(* CODESYS project Automatic stacking program.project

Project tree, tasks and I/O mapping:
  Device : CODESYS Control Win V3, 3S - Smart Software Solutions GmbH, order no. 305021, version 3.5.7.0
    application Application
      libraries: Standard, * (System)
      task MainTask (cyclic, interval t#20ms, priority 1) calls PLC_PRG
      task VISU_TASK (cyclic, interval 100 ms, priority 31) calls VisuElems.Visu_Prg
      program PLC_PRG [LD]
      visualisation Visualization
  text list GlobalTextList
*)

// Device/Application/PLC_PRG
PROGRAM PLC_PRG
VAR
	TON_01: TON;
	CTU_01: CTU;
	m2: BOOL;
	T: TIME;
	TT: WORD;
	stop: BOOL;
	start: BOOL;
	m1: BOOL;
	photo_sensor: BOOL;
END_VAR

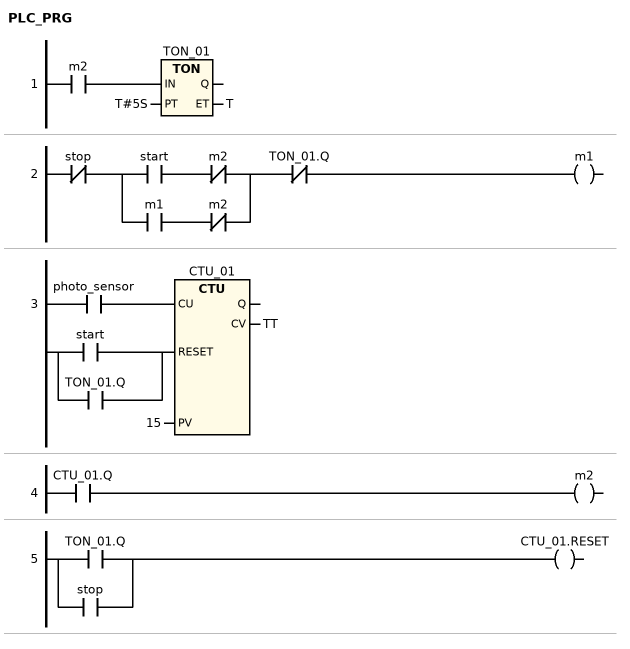
// NETWORK 1
TON_01(IN := m2, PT := T#5S, ET => T); // TON

// NETWORK 2
m1 := NOT stop AND (start AND NOT m2 OR m1 AND NOT m2) AND NOT TON_01.Q;

// NETWORK 3
CTU_01(CU := photo_sensor, RESET := start OR TON_01.Q, PV := 15, CV => TT); // CTU

// NETWORK 4
m2 := CTU_01.Q;

// NETWORK 5
CTU_01.RESET := TON_01.Q OR stop;

END_PROGRAM

// Device/Application/Visualization
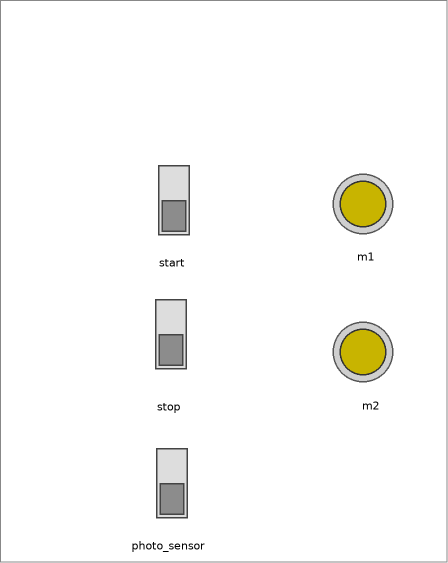
VISUALIZATION Visualization  // 448x563
    DipSwitch (139,165 70x70), variable: PLC_PRG.start, behaviour: TOGGLE, style: Switch-DipSwitch-Gray
    DipSwitch (136,299 70x70), variable: PLC_PRG.stop, behaviour: TOGGLE, style: Switch-DipSwitch-Gray
    DipSwitch (137,448 70x70), variable: PLC_PRG.photo_sensor, behaviour: TOGGLE, style: Switch-DipSwitch-Gray
    Lamp1 (328,169 70x70), variable: PLC_PRG.m1, style: Lamp-Lamp1-Yellow
    Lamp1 (328,317 70x70), variable: PLC_PRG.m2, style: Lamp-Lamp1-Yellow
    Label (97,248 150x30), "start"
    Label (291,242 150x30), "m1"
    Label (94,392 150x30), "stop"
    Label (296,391 150x30), "m2"
    Label (93,531 150x30), "photo_sensor"
END_VISUALIZATION
